// TIA Portal V18 export
FUNCTION "ST10Cyl_interface21-30" : Void   // FC1022, LAD
{ S7_Optimized_Access := 'FALSE' }
VERSION : 0.1
// stored: AutoNumber false, IsIECCheckEnabled false, SetENOAutomatically false, UDAEnableTagReadback false
   VAR_INPUT
      AlwaysON : Bool;
      E_stop : Bool;
   END_VAR
   VAR_TEMP
      tTest : Bool;
   END_VAR
BEGIN

REGION Network 1 (SCL): Cylinder 21-30 IO Interface (SCL)

   //Cylinder21 IO  H-shaftLiftingLiftingCylinder
   //Input
   "ST10Cylinder".Cy[21].In.WorkPositionSensor := "iH-shaftLiftingLiftingCylinderInWP" ;
   "ST10Cylinder".Cy[21].In.HomePositionSensor := "iH-shaftLiftingLiftingCylinderInHP" ;
   //Output
   "oH-shaftLiftingLiftingCylinderToWP" := "ST10Cylinder".Cy[21].Out.GoWorkPosition;
   "oH-shaftLiftingLiftingCylinderToHP" := "ST10Cylinder".Cy[21].Out.GoHomePosition;

   //Cylinder22 IO  H-shaftLiftingPalletLocationCylinder
   //Input
   "ST10Cylinder".Cy[22].In.WorkPositionSensor := "iH-shaftLiftingPalletLocationCylinderInWP" ;
   "ST10Cylinder".Cy[22].In.HomePositionSensor :="iH-shaftLiftingPalletLocationCylinderInHP"  ;
   //Output
   "oH-shaftLiftingPalletLocationCylinderToWP" := "ST10Cylinder".Cy[22].Out.GoWorkPosition;
   "oH-shaftLiftingPalletLocationCylinderToHP" := "ST10Cylinder".Cy[22].Out.GoHomePosition;

   //Cylinder23 IO  H-shaftLoadingStopperCylinder1
   //Input
   "ST10Cylinder".Cy[23].In.WorkPositionSensor := "oH-shaftLoadingStopperCylinder1_ToWP";
   "ST10Cylinder".Cy[23].In.HomePositionSensor := "oH-shaftLoadingStopperCylinder1_ToHP" ;
   //Output
   "oH-shaftLoadingStopperCylinder1_ToWP" := "ST10Cylinder".Cy[23].Out.GoWorkPosition;
   "oH-shaftLoadingStopperCylinder1_ToHP" := "ST10Cylinder".Cy[23].Out.GoHomePosition;

   //Cylinder24 IO  H-shaftLoadingStopperCylinder2
   //Input
   "ST10Cylinder".Cy[24].In.WorkPositionSensor := "oH-shaftLoadingStopperCylinder2_ToWP" ;
   "ST10Cylinder".Cy[24].In.HomePositionSensor := "oH-shaftLoadingStopperCylinder2_ToHP";
   //Output
   "oH-shaftLoadingStopperCylinder2_ToWP" := "ST10Cylinder".Cy[24].Out.GoWorkPosition;
   "oH-shaftLoadingStopperCylinder2_ToHP" := "ST10Cylinder".Cy[24].Out.GoHomePosition;

   //Cylinder25 IO  H-shaftLoadingStopperCylinder3
   //Input
   "ST10Cylinder".Cy[25].In.WorkPositionSensor := "oH-shaftLoadingStopperCylinder3_ToWP";
   "ST10Cylinder".Cy[25].In.HomePositionSensor := "oH-shaftLoadingStopperCylinder3_ToHP";
   //Output
   "oH-shaftLoadingStopperCylinder3_ToWP" := "ST10Cylinder".Cy[25].Out.GoWorkPosition;
   "oH-shaftLoadingStopperCylinder3_ToHP" := "ST10Cylinder".Cy[25].Out.GoHomePosition;

   //Cylinder26 H-shaftLoadingStopperCylinder4
   //Input
   "ST10Cylinder".Cy[26].In.WorkPositionSensor := "oH-shaftLoadingStopperCylinder4_ToWP";
   "ST10Cylinder".Cy[26].In.HomePositionSensor := "oH-shaftLoadingStopperCylinder4_ToHP" ;
   //Output
   "oH-shaftLoadingStopperCylinder4_ToWP" := "ST10Cylinder".Cy[26].Out.GoWorkPosition;
   "oH-shaftLoadingStopperCylinder4_ToHP" := "ST10Cylinder".Cy[26].Out.GoHomePosition;

   //Cylinder27 H-shaftTakeStopperCylinder1
   //Input
   "ST10Cylinder".Cy[27].In.WorkPositionSensor :="oH-shaftTakeStopperCylinder1_ToWP" ;
   "ST10Cylinder".Cy[27].In.HomePositionSensor :="oH-shaftTakeStopperCylinder1_ToHP";
   //Output
   "oH-shaftTakeStopperCylinder1_ToWP" :="ST10Cylinder".Cy[27].Out.GoWorkPosition;
   "oH-shaftTakeStopperCylinder1_ToHP" := "ST10Cylinder".Cy[27].Out.GoHomePosition;

   //Cylinder28 H-shaftTakeStopperCylinder2
   //Input
   "ST10Cylinder".Cy[28].In.WorkPositionSensor :="oH-shaftTakeStopperCylinder2_ToWP" ;
   "ST10Cylinder".Cy[28].In.HomePositionSensor := "oH-shaftTakeStopperCylinder2_ToHP";
   //Output
   "oH-shaftTakeStopperCylinder2_ToWP" := "ST10Cylinder".Cy[28].Out.GoWorkPosition;
   "oH-shaftTakeStopperCylinder2_ToHP" := "ST10Cylinder".Cy[28].Out.GoHomePosition;

   //Cylinder29 H-shaftTakeStopperCylinder3
   //Input
   "ST10Cylinder".Cy[29].In.WorkPositionSensor :="oH-shaftTakeStopperCylinder3_ToWP" ;
   "ST10Cylinder".Cy[29].In.HomePositionSensor :="oH-shaftTakeStopperCylinder3_ToHP";
   //Output
   "oH-shaftTakeStopperCylinder3_ToWP" := "ST10Cylinder".Cy[29].Out.GoWorkPosition;
   "oH-shaftTakeStopperCylinder3_ToHP" := "ST10Cylinder".Cy[29].Out.GoHomePosition;

    (*
    //Cylinder30 H-shaftLoadingStopperCylinder4_2  
   // //Input
   "ST10Cylinder".Cy[30].In.WorkPositionSensor := "oH-shaftLoadingStopperCylinder4_2";
   "ST10Cylinder".Cy[30].In.HomePositionSensor := NOT "oH-shaftLoadingStopperCylinder4_2";
   // //Output
    "oH-shaftLoadingStopperCylinder4_2" := "ST10Cylinder".Cy[30].Out.GoWorkPosition;
    "Feeding washer  lift Cylinder ToHP" := "ST10Cylinder".Cy[30].Out.GoHomePosition;
   *)
END_REGION

REGION Network 2: CY21 interface H-shaftLiftingLiftingCylinder
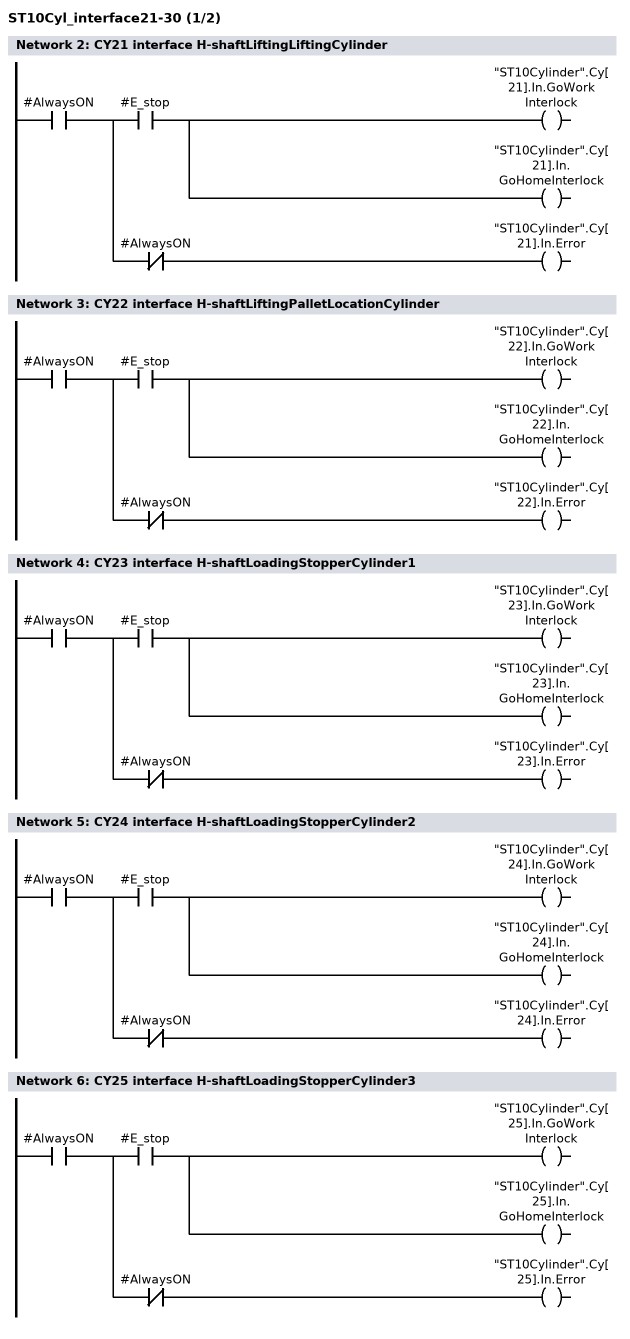
   RUNG wire#powerrail
      Contact( #AlwaysON )
      wire#w1
      Contact( #E_stop )
      wire#w2
      Coil( "ST10Cylinder".Cy[21].In.GoWorkInterlock )
   END_RUNG
   RUNG wire#w2
      Coil( "ST10Cylinder".Cy[21].In.GoHomeInterlock )
   END_RUNG
   RUNG wire#w1
      I_Contact( #AlwaysON )
      Coil( "ST10Cylinder".Cy[21].In.Error )
   END_RUNG
   // the same network as SCL:
   "ST10Cylinder".Cy[21].In.GoWorkInterlock := #AlwaysON AND #E_stop;
   "ST10Cylinder".Cy[21].In.GoHomeInterlock := #AlwaysON AND #E_stop;
   "ST10Cylinder".Cy[21].In.Error := #AlwaysON AND NOT #AlwaysON;
END_REGION

REGION Network 3: CY22 interface H-shaftLiftingPalletLocationCylinder
   RUNG wire#powerrail
      Contact( #AlwaysON )
      wire#w1
      Contact( #E_stop )
      wire#w2
      Coil( "ST10Cylinder".Cy[22].In.GoWorkInterlock )
   END_RUNG
   RUNG wire#w2
      Coil( "ST10Cylinder".Cy[22].In.GoHomeInterlock )
   END_RUNG
   RUNG wire#w1
      I_Contact( #AlwaysON )
      Coil( "ST10Cylinder".Cy[22].In.Error )
   END_RUNG
   // the same network as SCL:
   "ST10Cylinder".Cy[22].In.GoWorkInterlock := #AlwaysON AND #E_stop;
   "ST10Cylinder".Cy[22].In.GoHomeInterlock := #AlwaysON AND #E_stop;
   "ST10Cylinder".Cy[22].In.Error := #AlwaysON AND NOT #AlwaysON;
END_REGION

REGION Network 4: CY23 interface H-shaftLoadingStopperCylinder1
   RUNG wire#powerrail
      Contact( #AlwaysON )
      wire#w1
      Contact( #E_stop )
      wire#w2
      Coil( "ST10Cylinder".Cy[23].In.GoWorkInterlock )
   END_RUNG
   RUNG wire#w2
      Coil( "ST10Cylinder".Cy[23].In.GoHomeInterlock )
   END_RUNG
   RUNG wire#w1
      I_Contact( #AlwaysON )
      Coil( "ST10Cylinder".Cy[23].In.Error )
   END_RUNG
   // the same network as SCL:
   "ST10Cylinder".Cy[23].In.GoWorkInterlock := #AlwaysON AND #E_stop;
   "ST10Cylinder".Cy[23].In.GoHomeInterlock := #AlwaysON AND #E_stop;
   "ST10Cylinder".Cy[23].In.Error := #AlwaysON AND NOT #AlwaysON;
END_REGION

REGION Network 5: CY24 interface H-shaftLoadingStopperCylinder2
   RUNG wire#powerrail
      Contact( #AlwaysON )
      wire#w1
      Contact( #E_stop )
      wire#w2
      Coil( "ST10Cylinder".Cy[24].In.GoWorkInterlock )
   END_RUNG
   RUNG wire#w2
      Coil( "ST10Cylinder".Cy[24].In.GoHomeInterlock )
   END_RUNG
   RUNG wire#w1
      I_Contact( #AlwaysON )
      Coil( "ST10Cylinder".Cy[24].In.Error )
   END_RUNG
   // the same network as SCL:
   "ST10Cylinder".Cy[24].In.GoWorkInterlock := #AlwaysON AND #E_stop;
   "ST10Cylinder".Cy[24].In.GoHomeInterlock := #AlwaysON AND #E_stop;
   "ST10Cylinder".Cy[24].In.Error := #AlwaysON AND NOT #AlwaysON;
END_REGION

REGION Network 6: CY25 interface H-shaftLoadingStopperCylinder3
   RUNG wire#powerrail
      Contact( #AlwaysON )
      wire#w1
      Contact( #E_stop )
      wire#w2
      Coil( "ST10Cylinder".Cy[25].In.GoWorkInterlock )
   END_RUNG
   RUNG wire#w2
      Coil( "ST10Cylinder".Cy[25].In.GoHomeInterlock )
   END_RUNG
   RUNG wire#w1
      I_Contact( #AlwaysON )
      Coil( "ST10Cylinder".Cy[25].In.Error )
   END_RUNG
   // the same network as SCL:
   "ST10Cylinder".Cy[25].In.GoWorkInterlock := #AlwaysON AND #E_stop;
   "ST10Cylinder".Cy[25].In.GoHomeInterlock := #AlwaysON AND #E_stop;
   "ST10Cylinder".Cy[25].In.Error := #AlwaysON AND NOT #AlwaysON;
END_REGION

REGION Network 7: CY26 interface H-shaftLoadingStopperCylinder4
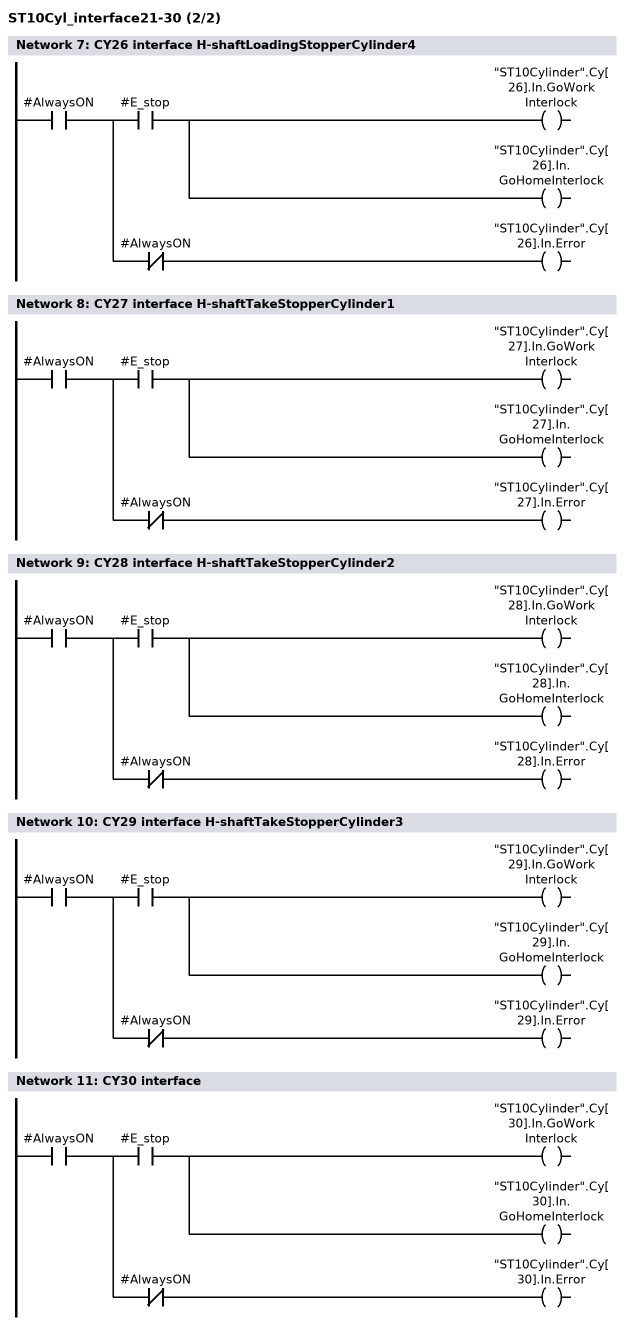
   RUNG wire#powerrail
      Contact( #AlwaysON )
      wire#w1
      Contact( #E_stop )
      wire#w2
      Coil( "ST10Cylinder".Cy[26].In.GoWorkInterlock )
   END_RUNG
   RUNG wire#w2
      Coil( "ST10Cylinder".Cy[26].In.GoHomeInterlock )
   END_RUNG
   RUNG wire#w1
      I_Contact( #AlwaysON )
      Coil( "ST10Cylinder".Cy[26].In.Error )
   END_RUNG
   // the same network as SCL:
   "ST10Cylinder".Cy[26].In.GoWorkInterlock := #AlwaysON AND #E_stop;
   "ST10Cylinder".Cy[26].In.GoHomeInterlock := #AlwaysON AND #E_stop;
   "ST10Cylinder".Cy[26].In.Error := #AlwaysON AND NOT #AlwaysON;
END_REGION

REGION Network 8: CY27 interface H-shaftTakeStopperCylinder1
   RUNG wire#powerrail
      Contact( #AlwaysON )
      wire#w1
      Contact( #E_stop )
      wire#w2
      Coil( "ST10Cylinder".Cy[27].In.GoWorkInterlock )
   END_RUNG
   RUNG wire#w2
      Coil( "ST10Cylinder".Cy[27].In.GoHomeInterlock )
   END_RUNG
   RUNG wire#w1
      I_Contact( #AlwaysON )
      Coil( "ST10Cylinder".Cy[27].In.Error )
   END_RUNG
   // the same network as SCL:
   "ST10Cylinder".Cy[27].In.GoWorkInterlock := #AlwaysON AND #E_stop;
   "ST10Cylinder".Cy[27].In.GoHomeInterlock := #AlwaysON AND #E_stop;
   "ST10Cylinder".Cy[27].In.Error := #AlwaysON AND NOT #AlwaysON;
END_REGION

REGION Network 9: CY28 interface H-shaftTakeStopperCylinder2
   RUNG wire#powerrail
      Contact( #AlwaysON )
      wire#w1
      Contact( #E_stop )
      wire#w2
      Coil( "ST10Cylinder".Cy[28].In.GoWorkInterlock )
   END_RUNG
   RUNG wire#w2
      Coil( "ST10Cylinder".Cy[28].In.GoHomeInterlock )
   END_RUNG
   RUNG wire#w1
      I_Contact( #AlwaysON )
      Coil( "ST10Cylinder".Cy[28].In.Error )
   END_RUNG
   // the same network as SCL:
   "ST10Cylinder".Cy[28].In.GoWorkInterlock := #AlwaysON AND #E_stop;
   "ST10Cylinder".Cy[28].In.GoHomeInterlock := #AlwaysON AND #E_stop;
   "ST10Cylinder".Cy[28].In.Error := #AlwaysON AND NOT #AlwaysON;
END_REGION

REGION Network 10: CY29 interface H-shaftTakeStopperCylinder3
   RUNG wire#powerrail
      Contact( #AlwaysON )
      wire#w1
      Contact( #E_stop )
      wire#w2
      Coil( "ST10Cylinder".Cy[29].In.GoWorkInterlock )
   END_RUNG
   RUNG wire#w2
      Coil( "ST10Cylinder".Cy[29].In.GoHomeInterlock )
   END_RUNG
   RUNG wire#w1
      I_Contact( #AlwaysON )
      Coil( "ST10Cylinder".Cy[29].In.Error )
   END_RUNG
   // the same network as SCL:
   "ST10Cylinder".Cy[29].In.GoWorkInterlock := #AlwaysON AND #E_stop;
   "ST10Cylinder".Cy[29].In.GoHomeInterlock := #AlwaysON AND #E_stop;
   "ST10Cylinder".Cy[29].In.Error := #AlwaysON AND NOT #AlwaysON;
END_REGION

REGION Network 11: CY30 interface
   RUNG wire#powerrail
      Contact( #AlwaysON )
      wire#w1
      Contact( #E_stop )
      wire#w2
      Coil( "ST10Cylinder".Cy[30].In.GoWorkInterlock )
   END_RUNG
   RUNG wire#w2
      Coil( "ST10Cylinder".Cy[30].In.GoHomeInterlock )
   END_RUNG
   RUNG wire#w1
      I_Contact( #AlwaysON )
      Coil( "ST10Cylinder".Cy[30].In.Error )
   END_RUNG
   // the same network as SCL:
   "ST10Cylinder".Cy[30].In.GoWorkInterlock := #AlwaysON AND #E_stop;
   "ST10Cylinder".Cy[30].In.GoHomeInterlock := #AlwaysON AND #E_stop;
   "ST10Cylinder".Cy[30].In.Error := #AlwaysON AND NOT #AlwaysON;
END_REGION
END_FUNCTION
